(* PLC project ifmCR711S_TemplateProject, CODESYS CODESYS V3.5 SP11 *)
(* stored: creationDateTime 2026-08-04T14:40:27.5703697, version 2.4.10.0, modificationDateTime 2026-08-04T14:25:20.5601505, organization ifm electronic *)
(* Project template with CR711S configured 2.25MByte Standard 2.25MByte Safety *)

PROGRAM LD_TEST
  VAR
    Sensor1 : BOOL;
    Sensor2 : BOOL;
    sensor3 : BOOL;
    PowerOn : BOOL;
    TON_0 : TON;
    CTU_0 : CTU;
    PowerOff : BOOL;
  END_VAR

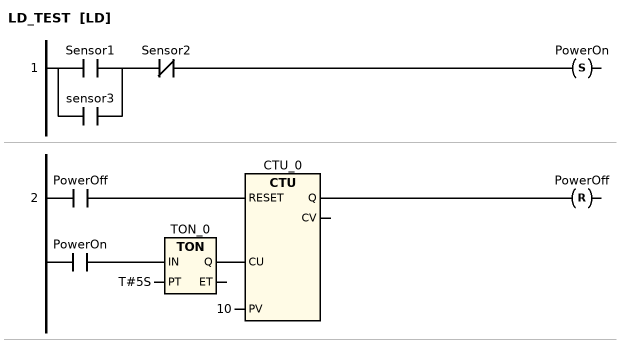
(* LD diagram, written out as Structured Text *)

IF (Sensor1 OR sensor3) AND NOT Sensor2 THEN PowerOn := TRUE; END_IF;
(* SECTION: safety interlocks *)


TON_0(IN := PowerOn, PT := T#5S);
CTU_0(CU := TON_0.Q, RESET := PowerOff, PV := 10);
IF CTU_0.Q THEN PowerOff := FALSE; END_IF;
END_PROGRAM
